PROGRAM MAIN
VAR
END_VAR

END_PROGRAM

(* stored: Version 1.1.0.1
   POU MAIN: Id {8462c308-cd40-4aaf-9c2d-c870f3576282} *)
